Staubli VAL3: _PA_grd_fin.pjx

--- _PA_grd_fin.pjx ---
Parameters version=s7.11.2 stackSize=5000 millimeterUnit=true
Program file=_alter_stauts.pgx
Program file=_finish.pgx
Program file=_Io.pgx
Program file=_mainLoop.pgx
Program file=_moveToScan.pgx
Program file=_recvFloat.pgx
Program file=_recvWaypoints.pgx
Program file=_sendJoint.pgx
Program file=_sendStatus.pgx
Program file=_startPass.pgx
Program file=_TmainLoop.pgx
Program file=Alter.pgx
Program file=start.pgx
Program file=stop.pgx
Data file=_PA_grd_fin.dtx

--- _PA_grd_fin.dtx ---
mdesc mNomSpeed = {tmax=25, rmax=25, blend=off}
bool bRunning
num nLastCmd
num nStatusSignal
num nWaypointCount
num nConnFlag
bool bMove
bool bAlterRun
num nAlterBegin
num nAlter
num nAlterEnd
public sio siTcpIpCommand = {link=Socket\Command}
public sio siTcpIpMotion = {link=Socket\Motion}
public sio siTcpIpFbk = {link=Socket\Feedback}
jointRx jHome = {j1=81.48, j2=37.87, j3=86.46, j4=-16.98, j5=-30.36, j6=14}
tool tTool = {x=225.4998, y=-0.0005, z=145.3992, ry=-90, fatherId=flange[0], ioLink=valve1}
mdesc mAlterspeed = {tmax=500, rmax=500}
trsf trOffset
public aio aiECAT1_0 = {link=EtherCAT-1\%IF0}
public dio doECAT1_192 = {link=EtherCAT-1\%Q192}
public aio aoECAT1_0 = {link=EtherCAT-1\%QF0}
public aio aoECAT1_32 = {link=EtherCAT-1\%QF32}
public aio aoECAT1_64 = {link=EtherCAT-1\%QF64}
public aio aoECAT1_96 = {link=EtherCAT-1\%QF96}
public aio aoECAT1_128 = {link=EtherCAT-1\%QF128}
public aio aoECAT1_160 = {link=EtherCAT-1\%QF160}
pointRx pCurent_pos = {fatherId=world[0]}
bool bAlterReset
num nDeltZ
num l_nHeight
pointRx pStart = {fatherId=world[0]}
pointRx pEnd = {fatherId=world[0]}
pointRx pApproach = {fatherId=world[0]}
pointRx pRetract = {fatherId=world[0]}
pointRx pWaypoints[100]
  [0] = {fatherId=world[0]}
  [1] = {fatherId=world[0]}
  [2] = {fatherId=world[0]}
  [3] = {fatherId=world[0]}
  [4] = {fatherId=world[0]}
  [5] = {fatherId=world[0]}
  [6] = {fatherId=world[0]}
  [7] = {fatherId=world[0]}
  [8] = {fatherId=world[0]}
  [9] = {fatherId=world[0]}
  [10] = {fatherId=world[0]}
  [11] = {fatherId=world[0]}
  [12] = {fatherId=world[0]}
  [13] = {fatherId=world[0]}
  [14] = {fatherId=world[0]}
  [15] = {fatherId=world[0]}
  [16] = {fatherId=world[0]}
  [17] = {fatherId=world[0]}
  [18] = {fatherId=world[0]}
  [19] = {fatherId=world[0]}
  [20] = {fatherId=world[0]}
  [21] = {fatherId=world[0]}
  [22] = {fatherId=world[0]}
  [23] = {fatherId=world[0]}
  [24] = {fatherId=world[0]}
  [25] = {fatherId=world[0]}
  [26] = {fatherId=world[0]}
  [27] = {fatherId=world[0]}
  [28] = {fatherId=world[0]}
  [29] = {fatherId=world[0]}
  [30] = {fatherId=world[0]}
  [31] = {fatherId=world[0]}
  [32] = {fatherId=world[0]}
  [33] = {fatherId=world[0]}
  [34] = {fatherId=world[0]}
  [35] = {fatherId=world[0]}
  [36] = {fatherId=world[0]}
  [37] = {fatherId=world[0]}
  [38] = {fatherId=world[0]}
  [39] = {fatherId=world[0]}
  [40] = {fatherId=world[0]}
  [41] = {fatherId=world[0]}
  [42] = {fatherId=world[0]}
  [43] = {fatherId=world[0]}
  [44] = {fatherId=world[0]}
  [45] = {fatherId=world[0]}
  [46] = {fatherId=world[0]}
  [47] = {fatherId=world[0]}
  [48] = {fatherId=world[0]}
  [49] = {fatherId=world[0]}
  [50] = {fatherId=world[0]}
  [51] = {fatherId=world[0]}
  [52] = {fatherId=world[0]}
  [53] = {fatherId=world[0]}
  [54] = {fatherId=world[0]}
  [55] = {fatherId=world[0]}
  [56] = {fatherId=world[0]}
  [57] = {fatherId=world[0]}
  [58] = {fatherId=world[0]}
  [59] = {fatherId=world[0]}
  [60] = {fatherId=world[0]}
  [61] = {fatherId=world[0]}
  [62] = {fatherId=world[0]}
  [63] = {fatherId=world[0]}
  [64] = {fatherId=world[0]}
  [65] = {fatherId=world[0]}
  [66] = {fatherId=world[0]}
  [67] = {fatherId=world[0]}
  [68] = {fatherId=world[0]}
  [69] = {fatherId=world[0]}
  [70] = {fatherId=world[0]}
  [71] = {fatherId=world[0]}
  [72] = {fatherId=world[0]}
  [73] = {fatherId=world[0]}
  [74] = {fatherId=world[0]}
  [75] = {fatherId=world[0]}
  [76] = {fatherId=world[0]}
  [77] = {fatherId=world[0]}
  [78] = {fatherId=world[0]}
  [79] = {fatherId=world[0]}
  [80] = {fatherId=world[0]}
  [81] = {fatherId=world[0]}
  [82] = {fatherId=world[0]}
  [83] = {fatherId=world[0]}
  [84] = {fatherId=world[0]}
  [85] = {fatherId=world[0]}
  [86] = {fatherId=world[0]}
  [87] = {fatherId=world[0]}
  [88] = {fatherId=world[0]}
  [89] = {fatherId=world[0]}
  [90] = {fatherId=world[0]}
  [91] = {fatherId=world[0]}
  [92] = {fatherId=world[0]}
  [93] = {fatherId=world[0]}
  [94] = {fatherId=world[0]}
  [95] = {fatherId=world[0]}
  [96] = {fatherId=world[0]}
  [97] = {fatherId=world[0]}
  [98] = {fatherId=world[0]}
  [99] = {fatherId=world[0]}
mdesc mAprSpeed = {tmax=10, rmax=10}
num i
mdesc mGrindSpeed = {tmax=10, rmax=10}
jointRx jScan = {j1=83.61, j2=38.15, j3=96.24, j4=-4.09, j5=-58.18, j6=-4.12}
num nByte
num nCmdSignal
num nForceTarget
num nX
num nY
num nZ
num nRx
num nRy
num nRz
num nKey
num x_nValue
public sio siTcpIpJoint = {link=Socket\Joint}
jointRx jCurrent
string l_sData

--- start.pgx ---
program start()
begin
  // ============================================================================
  // PA_grinding_V3 - TCP 통신 버전 (3 소켓)
  // Command (11001): ROS2 -> 로봇, 명령 수신
  // Motion (11000): ROS2 -> 로봇, Waypoint/Joint 데이터
  // Feedback (11002): 로봇 -> ROS2, 상태 송신
  // ============================================================================

  userPage()
  cls()
  putln("========================")
  putln("  PA_grinding_Started")
  putln("========================")
  putln("")

  // 초기화
  bRunning = true
  nLastCmd = 0
  nStatusSignal = 0
  nWaypointCount = 0
  nConnFlag = 0


  bMove=false
  bAlterRun=false
  nAlterBegin=0
  nAlter=0
  nAlterEnd=0

  // 소켓 타임아웃 설정 (non-blocking)
  sioCtrl(siTcpIpCommand, "timeout", 0)
  sioCtrl(siTcpIpMotion, "timeout", 0)
  sioCtrl(siTcpIpFbk, "timeout", 0)
  sioCtrl(siTcpIpJoint, "timeout", 0)

  // 버퍼 클리어
  clearBuffer(siTcpIpCommand)
  clearBuffer(siTcpIpMotion)
  clearBuffer(siTcpIpFbk)
  clearBuffer(siTcpIpJoint)

  putln("TCP 소켓 준비 완료")
  putln("  - Command: 11001 (수신)")
  putln("  - Motion: 11000 (수신)")
  putln("  - Feedback: 11002 (송신)")
  putln("  - Joint: 11003 (송신)")
  putln("")

  // 홈 위치로 이동

  putln("홈으로 이동 중")
  movej(jHome,tTool,mNomSpeed)
  waitEndMove()

  taskCreate "IO",50,_Io()
  taskCreate "Alter_status",50,_alter_stauts()
  cls()
  putln("========================")
  putln("      명령 대기 중...")
  putln("========================")
  putln("")
  putln("CMD: 1=종료, 2=스캔, 3=경로수신,")
  putln("     4=가공")


  // 메인 루프 태스크 시작
  taskCreate "mainLoop", 100, _mainLoop()

  // 메인 루프 종료 대기
  wait(taskStatus("mainLoop") == -1)

  cls()
  putln("PA_grindin 종료")

  // 홈 위치로 이동
  movej(jHome,tTool,mNomSpeed)
  waitEndMove()

end

--- _alter_stauts.pgx ---
program _alter_stauts()
begin
  while true
    gotoxy(0,12)
    put("* nAlter: "+toString("",nAlter)+"   ")
    gotoxy(12,12)
    put("* nAlterBegin: "+toString("",nAlterBegin)+"   ")
    delay(1)
  endWhile
end

--- _finish.pgx ---
program _finish()
begin
  // ============================================================================
  // CMD 1: 종료 - 홈 위치 복귀
  // ============================================================================
  cls()
  putln("[CMD 1] 종료 - 홈 복귀")
  nStatusSignal = 0
  call _sendStatus()

  movej(jHome, tTool, mNomSpeed)
  waitEndMove()

  putln("[CMD 1] 완료")
  bRunning = false

end

--- _Io.pgx ---
program _Io()
begin
  while true
    pCurent_pos=here(tTool[0],world)

    aioSet(aoECAT1_0,pCurent_pos[0].trsf.x)
    aioSet(aoECAT1_32,pCurent_pos[0].trsf.y)
    aioSet(aoECAT1_64,pCurent_pos[0].trsf.z)
    aioSet(aoECAT1_96,pCurent_pos[0].trsf.rx)
    aioSet(aoECAT1_128,pCurent_pos[0].trsf.ry)
    aioSet(aoECAT1_160,pCurent_pos[0].trsf.rz)

   if bAlterReset == true
      dioSet(doECAT1_192, 1)
      delay(0.1)
      bAlterReset= false
  else
  dioSet(doECAT1_192, 0)
  endIf

    nDeltZ=aioGet(aiECAT1_0)
    delay(0.004)
  endWhile
end

--- _mainLoop.pgx ---
program _mainLoop()
  local num l_nRetVal
begin
  // ============================================================================
  // 메인 루프 - Command 소켓에서 명령 수신
  // 명령: 1바이트 (1=종료, 2=스캔, 3=WP수신, 4=가공)
  // ============================================================================
  while bRunning

    // Command 소켓에서 명령 수신 (1바이트)
    l_nRetVal = sioGet(siTcpIpCommand, nByte)

    if l_nRetVal == 1
      // 데이터 수신됨
      nCmdSignal = nByte
      nConnFlag = 1
      putln("[CMD] 수신 = " + toString("", nCmdSignal))

      switch nCmdSignal
        case 1
          call _finish()
        break
        case 2
          call _moveToScan()
        break
        case 3
          call _recvWaypoints()
        break
        case 4
          call _startPass()
        break
        default
          putln("[WARN] 알 수 없는 명령: " + toString("", nCmdSignal))
        break
      endSwitch

      // Feedback 소켓으로 상태 응답 전송
      call _sendStatus()

    elseIf l_nRetVal == -1
      // 연결 끊김
      if nConnFlag == 1
        putln("[CMD] 연결 끊김")
        nConnFlag = 0
      endIf
    endIf

    delay(0.01)

  endWhile

end

--- _moveToScan.pgx ---
program _moveToScan()
begin
  // ============================================================================
  // CMD 2: 스캔 위치로 이동
  // ============================================================================
  cls()
  putln("* CMD "+ toString("", nCmdSignal) +": 스캔 위치로 이동")

  nStatusSignal = 0
  call _sendStatus()

  movej(jScan, tTool, mNomSpeed)
  waitEndMove()
  gotoxy(0,1)
  putln("* 스캔 위치 도달")

  call _sendJoint()

  nStatusSignal = 2
  call _sendStatus()

  gotoxy(0,8)
  putln("현재 상태값 : "+ toString("", nStatusSignal))
  putln("========================")
  putln("      명령 대기 중...")
  putln("========================")
end

--- _recvWaypoints.pgx ---
program _recvWaypoints()
  local num l_nJ1
  local num l_nJ2
  local num l_nJ3
  local num l_nJ4
  local num l_nJ5
  local num l_nJ6
begin
  // ============================================================================
  // CMD 3: 웨이포인트 수신 (TCP - Motion 소켓)
  // 데이터: DOC(float) + Force(float) + Count(float) + Joints(6 floats each)
  // Joint: j1, j2, j3, j4, j5, j6 (degrees)
  // ============================================================================
  cls()
  putln("* CMD "+ toString("", nCmdSignal) +":  웨이포인트 수신 시작")
  nStatusSignal = 0

  // Count 수신
  call _recvFloat(nWaypointCount)
  nWaypointCount = roundDown(nWaypointCount)
  gotoxy(0,1)
  putln("  Count=" + toString("", nWaypointCount))

  // 각 Waypoint 수신 (6축 Joint)
  for i = 0 to nWaypointCount - 1
    call _recvFloat(nX)
    call _recvFloat(nY)
    call _recvFloat(nZ)

    pWaypoints[i].trsf.x = nX
    pWaypoints[i].trsf.y = nY
    pWaypoints[i].trsf.z = nZ
    pWaypoints[i].trsf.rx = -5
    pWaypoints[i].trsf.ry = 0
    pWaypoints[i].trsf.rz = 90

    if i == 0 or  i == nWaypointCount - 1
      putln("  P[" + toString("", i) + "]=" + toString("", nX) + "," + toString("", nY) + "," + toString("", nZ) + "," + toString("", nRx) + "," + toString("", nRy) + "," + toString("", nRz))
    endIf
  endFor

  gotoxy(0,4)
  putln("* 웨이 포인트 수신 완료")
  nStatusSignal = 3
  call _sendStatus()

  gotoxy(0,8)
  putln("현재 상태값 : "+ toString("", nStatusSignal))
  putln("========================")
  putln("      명령 대기 중...")
  putln("========================")
end

--- _sendJoint.pgx ---
program _sendJoint()
begin
  jCurrent = herej()

  sioSet(siTcpIpJoint, jCurrent.j1)
  sioSet(siTcpIpJoint, jCurrent.j2)
  sioSet(siTcpIpJoint, jCurrent.j3)
  sioSet(siTcpIpJoint, jCurrent.j4)
  sioSet(siTcpIpJoint, jCurrent.j5)
  sioSet(siTcpIpJoint, jCurrent.j6)
end

--- _sendStatus.pgx ---
program _sendStatus()
  local num l_nData
begin
  // ============================================================================
  // 상태 응답 전송 (1바이트)
  // 0=Idle, 1=Ready, 2=PassDone, 3=Error
  // ============================================================================

  l_nData = nStatusSignal
  sioSet(siTcpIpFbk, l_nData)

  putln("[TCP] STATUS = " + toString("", nStatusSignal))

end

--- _startPass.pgx ---
program _startPass()
begin
  cls()
  putln("* CMD "+ toString("", nCmdSignal) +": 가공 시작")

  if taskStatus("alter")!=1
    taskCreate "alter",100,Alter()
  endIf

  // Approach/Retract 높이 설정 (mm)
  l_nHeight = 5

  // 시작점, 끝점의 직교좌표 계산
  pStart = pWaypoints[0]
  pEnd =  pWaypoints[nWaypointCount - 1]

  // Approach 포인트 (시작점 위)
  pApproach = pStart
  pApproach.trsf.z = pApproach.trsf.z + l_nHeight

  // Retract 포인트 (끝점 위)
  pRetract = pEnd
  pRetract.trsf.z = pRetract.trsf.z + l_nHeight

  // 1. Approach 위치로 이동
  gotoxy(0,1)
  putln("  [1] Approach 이동 (Z+" + toString("", l_nHeight) + ")")
  alterMovel(pApproach, tTool, mNomSpeed)
  waitEndMove()

  // 2. 시작점으로 하강
  gotoxy(0,2)
  putln("  [2] 시작점 하강")
  alterMovel(pStart, tTool, mAprSpeed)
  waitEndMove()
  bAlterRun = true

  // 3. 가공 경로 실행
  gotoxy(0,3)
  putln("  [3] 그라인딩 시작")
  for i = 0 to nWaypointCount - 1
    bAlterReset=true
    alterMovel(pWaypoints[i], tTool, mGrindSpeed)
    waitEndMove()

    // TODO: Force Control 적용
  endFor
  alterEnd()
  bAlterRun=false
  nAlter=0
  nAlterBegin=0
  taskKill("alter")

  // 4. Retract 위치로 상승
  gotoxy(0,4)
  putln("  [4] Retract 이동 (Z+" + toString("", l_nHeight) + ")")
  alterMovel(pRetract, tTool, mAprSpeed)
  waitEndMove()

  gotoxy(0,5)
  putln("* 그라인딩 완료")
  nStatusSignal = 4
  call _sendStatus()

  gotoxy(0,8)
  putln("현재 상태값 : "+ toString("", nStatusSignal))
  putln("========================")
  putln("      명령 대기 중...")
  putln("========================")
end

--- _TmainLoop.pgx ---
program _TmainLoop()
begin
  cls()
  putln("[키보드 명령]")
  putln("  F1 = 종료")
  putln("  F2 = 스캔위치 이동")
  putln("  F3 = 웨이포인트 수신")
  putln("  F4 = 가공 시작")
  putln("")

  while bRunning

    nKey = get()

    switch nKey
      case 271
        nCmdSignal = 1
        putln("[F1] 종료")
      break
      case 272
        nCmdSignal = 2
        putln("[F2] 스캔 이동")
      break
      case 273
        nCmdSignal = 3
        putln("[F3] 웨이포인트 수신")
      break
      case 274
        nCmdSignal = 4
        putln("[F4] 가공 시작")
      break
      default
        nCmdSignal = 0
      break
    endSwitch

    if nCmdSignal != 0
      switch nCmdSignal
        case 1
          call _finish()
        break
        case 2
          call _moveToScan()
        break
        case 3
          call _recvWaypoints()
        break
        case 4
          call _startPass()
        break
      endSwitch

      // 상태 응답 전송
      //call _sendStatus()

      gotoxy(0,9)
      putln("다음 명령 대기 (F1~F4)...")
      nCmdSignal = 0
    endIf

    delay(0.01)

  endWhile

end

--- Alter.pgx ---
program Alter()
begin
  wait(bAlterRun == true and isSettled() == false)
  nAlterBegin=alterBegin(world,mAlterspeed)

  while nAlterBegin>=0 and bAlterRun==true
    if bAlterRun==true
      trOffset.x = 0
      trOffset.y = 0
      trOffset.z = nDeltZ
      trOffset.rx = 0
      trOffset.ry = 0
      trOffset.rz = 0
    elseIf bAlterRun==false
      trOffset.z = 0
    endIf
    nAlter = alter(trOffset)
      delay(0.004)
  endWhile
end
